TYPE ST_ParamFixed :
STRUCT
END_STRUCT
END_TYPE

(* stored: Version 1.1.0.1, ProductVersion 3.1.4020.6
   DUT ST_ParamFixed: Id {5762a14a-76f3-4b2b-8386-4034caf55c9a} *)
